FUNCTION F_SV_Daten_Schreiben : BOOL
VAR_IN_OUT
	Stellwert_Stellung	: BOOL;
END_VAR
VAR_INPUT
	Stellwert		: ST_SV_Stellwert;
END_VAR
VAR
END_VAR

Stellwert_Stellung := Stellwert.Stellung;

END_FUNCTION

(* stored: Version 1.1.0.1, ProductVersion 3.1.4024.9
   POU F_SV_Daten_Schreiben: Id {aa7fbdb7-59ae-4f8c-98ad-47d7c767b39b}, SpecialFunc None *)
